TYPE T_TimeLog : STRING[15];
END_TYPE

(* stored: Version 1.1.0.1
   DUT T_TimeLog: Id {368da0de-f011-4578-9620-a11eff12e12e} *)
